TYPE "PLCtoMES_PrintExchange"
VERSION : 0.1
   STRUCT
      "P-PrintReq" : Bool;
      "P-PrintPartID" : Array[1..10] of String[48];
      Reserve : Array[1..498] of Byte;
   END_STRUCT;

END_TYPE

